FUNCTION_BLOCK PAClassAlarmingBase EXTENDS ACComponent
VAR_INPUT
END_VAR
VAR_OUTPUT
END_VAR
VAR
END_VAR

END_FUNCTION_BLOCK

(* stored: Version 1.1.0.1, ProductVersion 3.1.4020.12
   POU PAClassAlarmingBase: Id {17c5b712-7c4d-410f-bfb8-3d09306de874}, SpecialFunc None *)
